{attribute 'linkalways'} 
{attribute 'no_explicit_call' := 'This FB is a CLASS and must be accessed using methods or properties'}
{attribute 'enable_dynamic_creation'}
FUNCTION_BLOCK Node_ContainerType_Vector_TcVnDMatch EXTENDS Node
VAR
    out : _GUID;
END_VAR

METHOD PUBLIC  Clone : I_Node
VAR
	pNode : POINTER TO Node_ContainerType_Vector_TcVnDMatch;
END_VAR
pNode := __NEW(Node_ContainerType_Vector_TcVnDMatch);
Clone := pNode^;
END_METHOD

METHOD FB_init : BOOL
VAR_INPUT
	bInitRetains : BOOL; // if TRUE, the retain variables are initialized (warm start / cold start)
	bInCopyCode : BOOL;  // if TRUE, the instance afterwards gets moved into the copy code (online change)
END_VAR
AddOutput('out', out);
END_METHOD

METHOD PROTECTED OnExecute
out.Value := ContainerType_Vector_TcVnDMatch;
END_METHOD

END_FUNCTION_BLOCK

(* stored: Version 1.1.0.1, ProductVersion 3.1.4026.17
   POU Node_ContainerType_Vector_TcVnDMatch: Id {737c7d37-8e48-0a0b-2f5e-e03715e852ea}, SpecialFunc None
   Folder Constructor: Id {e95eba1b-008c-01d1-00c4-4c02b19e649d}
   Method Clone: Id {56d1cb28-be46-078d-19c3-23e7dea82eb6}
   Method FB_init: Id {adf47681-b61e-0305-06ba-b1be5930a2ff}
   Method OnExecute: Id {b3f3d274-440c-0009-33c6-e77b8b7053bf} *)
